(* IEC 61131-3 sources: CodesysTest/alpha/export/PackML/OMAC/GlobalConstants, 1 file *)

(* ---- PackML_Omac_GVL.gvl.st ---- *)
(*#-#-#-#-#-#-#-#-#-#---Declaration---#-#-#-#-#-#-#-#-#-#-#-#-#*)

VAR_GLOBAL CONSTANT
	gc_usiMaxModes: USINT := 10;	// Maximum number of unit modes.
END_VAR
